--- timerDialog.pgx ---
public program timerDialog(screen& x_scr, string x_sMsg, num x_nTime)
  local num l_nTime
  local num l_nStartLine
  local num l_nLine
  local num i
  local string l_sMessage
begin
  //-----------------------------------------------------------------------
  //Header begin
  //Description of program
  //  Displays a dialog box from the data message. After called this program,
  //  you will regenerate your interface.
  // 从数据消息中显示一个对话窗口。在call这个程序后，你可以再生你的界面。
  //Input parameters
  //  string x_sMsg :
  //    role : Message that you want to display
  //    作用：你想去展示的消息。
  //  num x_nTime :
  //    role : Waiting time before restoring the main
  //   作用：在存储主界面后，等待的时间
  //Example
  //  call timerDialog(scrMy,"Hello",2)
  //
  //History
  //  Creation : 28-04-08 - f.Rob
  //Header end
  //-----------------------------------------------------------------------
  //Use for other task
  //If "timerDialog" is already used, put a message error and return in
  //the calling program
  //如果"计时器窗口" 已经被使用，弹出一个消息错误，然后回到calling该程序。
  if watch(bShowDialog==false,2)==false
    bShowDialog=false
    logMsg("Error dialog resoursing")
    return
  else
    setMutex(bShowDialog)
    //Start clock  开始计时
    l_nTime=clock()
    //Copy all the values from the first element to the second one
    // 复制所有的值从第一个元素到第二个元素
    call stringCopy(x_sMsg,sMessage)
    //Divide the message if it is too long (Search a space for cut the message)
    //如果消息太长，把它进行分割（以空格为标志来分割消息）
    //Return the numbers of lines used for writing the message.
    //返回用来写消息的行数目。
    call divideString(sMessage,l_nLine)
    l_nStartLine=round(5-l_nLine/2)
    do
      //Start Line
      call type(x_scr,0,l_nStartLine-2,"┌──────────────────────────────────────┐")
      call type(x_scr,0,l_nStartLine-1,"│                                      │")
      //Write the message
      for i=0 to l_nLine
        call type(x_scr,0,l_nStartLine+i,"")
        call type(x_scr,39,l_nStartLine+i,"")
        l_sMessage=sMessage[i]
        //Displays the message in center of the box
        call typeCenter(x_scr,i+l_nStartLine,l_sMessage,38,false)
        call type(x_scr,0,l_nStartLine+i,"│"+l_sMessage+"│")
      endFor
      //End Line
      call type(x_scr,0,l_nStartLine+l_nLine+1,"│                                      │")
      call type(x_scr,0,l_nStartLine+l_nLine+2,"└──────────────────────────────────────┘")
      //Release
      if x_nTime==0
        delay(0.1)
      else
        delay(0)
      endIf
      //Waiting time
    until (clock()-l_nTime)>=x_nTime
    //Reset the variables
    bShowDialog=false
    //global variable : Indicates that you want refresh the screen
    bUseRefresh=true
    delay(0)
  endIf
end

--- type.pgx ---
public program type(screen& x_scr, num x_nX, num x_nY, string x_sMessage)
begin
  //-----------------------------------------------------------------------
  //Header begin
  //Description of program
  //  Displays one string to pX column
  //  and pY Line.
  // 显示一个字符串到pX列，pY行。
  //Input parameters
  //  num x_nX :
  //    role : Cursor column
  //    作用：光标列
  //  num x_nY :
  //    role : Cursor row
  //    作用：光标行
  //  string x_sMessage :
  //    role : Message that you want to display
  //   作用：你想去显示的消息
  //Example
  //  call type(scrMy,2,5,"Staubli)
  //
  //History
  //  Creation : 28-04-08 - f.Rob
  //
  //  Modified : 22 Aug 2011 - J. Cook  Added user screens
  //Header end
  //-----------------------------------------------------------------------
  gotoxy(x_scr, x_nX,x_nY)
  put(x_scr, x_sMessage)
end

--- typeCenter.pgx ---
public program typeCenter(screen& x_scr, num x_nY, string& x_sMessage[], num x_nLength, bool x_bShow)
  local num l_nX
  local num l_nLenMess
  local string l_sMessage
  local num i
begin
  //-----------------------------------------------------------------------
  //Header begin
  //Description of program
  //  Displays one message in center and at the Y position of the userPage.
  //  - If x_bShow is true : if the length of the message is greater than
  //  x_nLength it will be truncated.
  //  显示一条消息在中间和在用户界面的Y位置。
  //  如果x_bShow是真值：如果消息的长度是大于长度x_nLength，这将会被截断。
  //  - If x_bShow is false : if the length of the message is less than
  //  如果x_bShow是假值：如果消息的长度是小于长度x_nLength，字符会被空格替代，否则消息会被截断。
  //  x_nLength,the characters are replaced by spaces otherwise the message
  //  will be truncated.
  //
  //Input parameters
  //  num x_nY :
  //    role : cursor row  作用：光标行
  //  num x_nLength :
  //    role : max lenght of the message  作用：消息的最大长度
  //  bool x_bShow :
  //    role : set to true if you just want to display a message and false if
  //   作用:如果你仅仅想去显示一条消息，就设为真值；如果你想在消息的前面或后面插入空格，那就设为假值。
  //    you want to add spaces before and after the message.
  //
  //Output parameters
  //  string x_sMessage :
  //    role : Message that you want to display. It can be modified by
  //    作用：你想去显示的消息。当你想要在消息的前面或后面插入空格，可以修改程序。
  //    the program when you want add spaces before and after the message
  //
  //Example
  //  call typeCenter(scrMy,5,"Hello",10,true) //Displays "Hello" in the middle of the line 5
  //
  //History
  //  Creation : 28-04-08 - f.Rob
  //
  //  Modified : 08-08-22 - J.Cook     Add screen parameter
  //Header end
  //-----------------------------------------------------------------------
  l_nLenMess=getDisplayLen(x_sMessage)
  if (l_nLenMess>x_nLength)
    //Comprime
    call strlength(x_sMessage,x_nLength)
    //Found the pos to start write
    l_nX=20-(x_nLength/2)
  else
    //Found the pos to start write
    l_nX=20-(l_nLenMess/2)
  endIf
  l_sMessage=x_sMessage
  if x_bShow
    //You want to display your message
    call type(x_scr, l_nX,x_nY,l_sMessage)
  else
    //Put spaces before the message
    for i=0 to max(l_nX-(40-x_nLength)/2,0)-1
      l_sMessage=" "+l_sMessage
    endFor
    //Put spaces after the message and give it
    call strFill(l_sMessage,x_nLength,x_sMessage)
  endIf
end

--- typeLen.pgx ---
public program typeLen(screen& x_scr, num x_nX, num x_nY, string x_sMessage, num x_nLength)
begin
  //-----------------------------------------------------------------------
  //Header begin
  //Description of program
  //  Displays one message to pX column and pY Line. 显示一条消息到pX列，pY行。
  //  If the length of the message is less than x_nLen, the characters are replaced
  //  by spaces otherwise the message will be truncated.
  //  如果消息的长度是少于长度x_nLen，字符将被空格替代，否则消息会被截断。
  //Input parameters
  //  num x_nX :
  //    role : cursor column  作用：光标列
  //  num x_nY :
  //    role : cursor row     作用：光标行
  //  string x_sMessage :
  //    role : message that you want to display  作用：你想要去显示的消息
  //  num x_nLength :
  //    role : max length of the message  作用：消息的最大长度
  //
  //Example
  //  call typeLen(scrMy,2,5,"Hello",10)
  //
  //History
  //  Creation : 28-04-08 - f.Rob
  //
  //  Modified : 22 Aug 2011 - J. Cook  Added user screens
  //Header end
  //-----------------------------------------------------------------------
  call strlength(x_sMessage,x_nLength)
  call type(x_scr,x_nX,x_nY,x_sMessage)
end

--- typeMenu.pgx ---
public program typeMenu(screen& x_scr, num x_nKeyFct, string x_sMessage)
  local string l_sMessage
  local string l_sMessEmpty
  local num l_nMaxLen
  local num l_nPosX
  local num l_nPosY
  local num l_nStep
  local num l_nI
begin
  //-----------------------------------------------------------------------
  //Header begin
  //Description of program
  //  Displays the message x_sMessage (4 characters max otherwise it will be
  //  truncated)in the userPage above the functions keys F1 to F8 (1 to 8).
  //  显示用户界面上功能键F1到F8的消息x_sMessage（最多4个字符，否则将会被截断）
  //Input parameters
  //  num x_nKeyFct :
  //    role : function key that you want to display
  //    作用：你想要去显示的功能键
  //    possible values : 1 to 8 (there are 8 functions keys : F1 to F8)
  //    有可能的值：1到8（存在8个功能键：F1到F8）
  //  string x_sMessage :
  //    role : Message that you want to display
  //   作用：你想要去显示的消息
  //Examples
  //  call typeMenu(scrMy,1,"Informations") //Displays "Inf." above the F1 key
  //  call typeMenu(scrMy,5,"List Simple") //Displays "List" above the F5 key
  //
  //History
  //  Creation : 28-04-08 - f.Rob
  //
  //  Modified : 08-08-22 - J.Cook     Add screen parameter
  //Header end
  //-----------------------------------------------------------------------
  l_nStep=5
  l_nPosY=13
  l_sMessEmpty="     "
  if (x_nKeyFct>=1) and (x_nKeyFct<=8)
    l_nMaxLen=4
    //Control the length of x_sMessage
    //Europe case
    if (getDisplayLen(x_sMessage)>l_nMaxLen)
      if len(x_sMessage)==getDisplayLen(x_sMessage)
        //Find a space in the message
        l_nI=find(x_sMessage," ")
        if l_nI<5 and l_nI>2
          //Take only characters before spaces
          l_sMessage=mid(x_sMessage,l_nI,0)
        else
          //Delete characters after the l_nMaxLen-1 and add a point (.) at the end.
          l_sMessage=mid(x_sMessage,l_nMaxLen-1,0)
          l_sMessage=l_sMessage+"."
        endIf
      else
        //Asia one
        l_sMessage=mid(x_sMessage,2,0)
      endIf
    else
      l_sMessage=x_sMessage
    endIf
    //Position X
    l_nPosX=(x_nKeyFct-1)*l_nStep+1
    //Control the length of l_sMessage and cut it if it's too long
    call strFill(l_sMessage,4,l_sMessage)
    //Displays l_sMessage to l_nPosX column and l_nPosY Line
    call type(x_scr, l_nPosX,l_nPosY,l_sMessage)
  endIf
end
